PROGRAM Axis_Template
VAR

END_VAR

//Initial parameters of an Axis
(*IF _TaskInfo[fbGetCurTaskIndex.index].FirstCycle THEN
    //Initial default values:
    GVL.astAxes[1].stControl.fVelocity := GVL.astAxes[1].stConfig.fVelocityDefaultSlow;
    GVL.astAxes[1].stConfig.eHomeSeq := 0;
    GVL.astAxes[1].stConfig.fHomePosition := 0.0;
    GVL.astAxes[1].stConfig.fHomeFinishDistance := 0.0;
END_IF*)

//Define ACTIONS() or write exclusive code for an specific axis.
//Eg. Stop when temperature reaches certain values, reduce speed if  a signal is activated, etc.

END_PROGRAM

(* stored: Version 1.1.0.1, ProductVersion 3.1.4024.5
   POU Axis_Template: Id {1a43acb4-bd2e-4637-97fb-9976d47292b6}, SpecialFunc None *)
